// TIA Portal V20 export
// export: Created 2025-12-01T14:56:15.9263385Z, ExportSetting None, DisplayName Totally Integrated Automation Portal, DisplayVersion V20 Update 3, DisplayName TIA Portal Openness, DisplayVersion V20 Update 3, DisplayName TIA Portal Version Control Interface, DisplayVersion V20 Update 3, DisplayName STEP 7 Professional, DisplayVersion V20 Update 3, DisplayName STEP 7 Safety, DisplayVersion V20 Update 2, DisplayName WinCC Basic/Comfort/Advanced, DisplayVersion V20 Update 3, DisplayName WinCC Professional, DisplayVersion V20 Update 3, DisplayName WinCC Unified, DisplayVersion V20 Update 3
TYPE "ROUT_Destino_Desvios"
   STRUCT
      Destino : UInt;   // Destino de la Etiqueta
      Desvios : Array[0.."ROUT_Num_Max_Desvios"] of Struct   // Desvios por las Etiquetas
         SCR : UInt;   // Numero de SCR
         Bits : Byte;   // Bits a Activar
         Libre : Byte;   // Byte libre para opciones a añadir en la estructura sin que crezca
      END_STRUCT;
   END_STRUCT;
   // Desvios[0..20].Bits := B#16#01;
END_TYPE
